(* CoDeSys 2.3.9.42 project: CR0451 AGV.pro *)
(* Libraries: ifm_PDMsmart_util_V010007.lib 26.10.09 12:29:10, ifm_RAWCan\ifm_RAWCan_NT_V020004.lib 3.11.15 19:07:52, ifm_J1939_NT\ifm_J1939_NT_V020004.lib 18.9.14 16:13:02, Util.lib 6.11.07 16:39:24, SysLibPlcCtrl.lib 13.6.03 15:49:00, SysLibFile.lib 23.9.04 10:11:36, SysLibTime.lib 27.4.05 10:36:52, LinuxSystemLib.Lib 18.3.03 13:26:50, ifm_pdm_file_V010006.lib 14.1.08 14:21:32, standard.lib 4.10.05 11:14:46, SysLibVisuBasicDisplay.lib 22.3.17 09:59:30, SysLibTargetVisu.lib 5.4.04 13:31:00, SysLibCallback.lib 26.9.08 17:43:52, ifm_CR0451_callback_visu.lib 22.3.17 09:59:30, SysLibStr.lib 13.6.03 15:49:00, ifm_CR0451\ifm_CR0451_Init_V030000.lib 22.3.17 09:59:30 *)

(* PLC configuration (modules and I/O channels)
Device Configuration [LocalConfiguration] node 0, in %IB0 out %QB0 {IFM_PARAM_WORD_TIME = 10}
KEY_F1 AT %IB0 [ChInputBool] F1 Key
KEY_F2 AT %IB1 [ChInputBool] F2 Key
KEY_F3 AT %IB2 [ChInputBool] F3 Key
KEY_F4 AT %IB3 [ChInputBool] F4 Key
KEY_UP AT %IB4 [ChInputBool] Up Key
KEY_DOWN AT %IB5 [ChInputBool] Down Key
KEY_LEFT AT %IB6 [ChInputBool] Left Key
KEY_RIGHT AT %IB7 [ChInputBool] Right Key
KEY_OK AT %IB8 [ChInputBool] Ok Key
RT_F1 AT %IB9 [ChInputBool] Rising Edge F1 Key
RT_F2 AT %IB10 [ChInputBool] Rising Edge F2 Key
RT_F3 AT %IB11 [ChInputBool] Rising Edge F3 Key
RT_F4 AT %IB12 [ChInputBool] Rising Edge F4 Key
RT_UP AT %IB13 [ChInputBool] Rising Edge Up Key
RT_DOWN AT %IB14 [ChInputBool] Rising Edge Down Key
RT_LEFT AT %IB15 [ChInputBool] Rising Edge Left Key
RT_RIGHT AT %IB16 [ChInputBool] Rising Edge Right Key
RT_OK AT %IB17 [ChInputBool] Rising Edge Ok Key
FT_F1 AT %IB18 [ChInputBool] Falling Edge F1 Key
FT_F2 AT %IB19 [ChInputBool] Falling Edge F2 Key
FT_F3 AT %IB20 [ChInputBool] Falling Edge F3 Key
FT_F4 AT %IB21 [ChInputBool] Falling Edge F4 Key
FT_UP AT %IB22 [ChInputBool] Falling Edge Up Key
FT_DOWN AT %IB23 [ChInputBool] Falling Edge Down Key
FT_LEFT AT %IB24 [ChInputBool] Falling Edge Left Key
FT_RIGHT AT %IB25 [ChInputBool] Falling Edge Right Key
FT_OK AT %IB26 [ChInputBool] Falling Edge Ok Key
Key Events [KeyEvents] node 3, in %IB27 out %QB0
  KEY_CHANGED AT %IB27 [ChInputBool] Event: Key Changed
  KEY_PRESSED AT %IB28 [ChInputBool] Event: Key is pressed
SUPPLY_VOLTAGE_VBBS AT %IW15 [ChInputWord] Supply voltage VBBS
SUPPLY_VOLTAGE_VU AT %IW16 [ChInputWord] Supply voltage VU
TEMPERATURE AT %IW17 [ChInputInt] Temperature
SCREEN_BACKLIGHT_CTRL AT %QB0 [ChOutputByte] Screen Backlight (0 - 100%)
KEY_BACKLIGHT_CTRL AT %QB1 [ChOutputByte] Key Backlight (0 - 100%)
CANopen Interface [CAN_OPEN] node 0, in %IB36 out %QB2
J1939 Interface [CAN_J1939] node 1, in %IB36 out %QB2
*)

(* Global variable list: Variables_Globales *)
VAR_GLOBAL

(* var for page and item menu selection *)
	menu_glob: INT:=1;
	PageIntern: WORD;
	Actual_Page: WORD;
  menu_item: ARRAY [0..20] OF BOOL;



END_VAR

VAR_GLOBAL RETAIN

END_VAR

(* POU PLC_PRG, ST *)
PROGRAM PLC_PRG
VAR
      xInitPageControl: BOOL;
	Shift_on_page_P00100: Shift_on_page_P00xxx;
	Shift_on_page_P00101: Shift_on_page_P00xxx;
	Shift_on_page_P00102: Shift_on_page_P00xxx;
	Shift_on_page_P00103: Shift_on_page_P00xxx;
	CAN_ENABLE_CAN1: CAN_ENABLE;
END_VAR
(* -++++++++++++++++-hieronder kun je het CAN channel activeren met   CAN_ENABLE  en/of  J1939_ENABLE-++++++++*)
CAN_ENABLE_CAN1(ENABLE:=TRUE, CHANNEL:= 1, BAUDRATE:=500 , RESULT=> );


(*++++++++++++++++++++++++++++++++++++++++++++++++++++++++++++++++++++++++++++++++++++++++++*)
(* -------------------------------------------initialiseren van het display CR0451---------------------------------------------------------------- *)
BasicDisplay_Init();
PDM_PAGECONTROL(
	INIT:= xInitPageControl,
	INIT_PAGE:=00001 ,
	PAGE_UP:= ,
	PAGE_DOWN:= ,
	PAGE_EXTERN:=PageIntern ,
	PAGE_MAX:=00108 ,                       (* de "hoogste pagina nummer opgeven*)
	BASENAME:='P',
	ACT_PAGE=>Actual_Page );

xInitPageControl:=FALSE;  (* pdm_pagecontrol moet slechts 1 keer worden uitgevoerd bij opstart, daarom init onmiddellijk op False gezet *)

(* startpagina en achterliggende pagina's beheren *)
(* zie eigen aangemaakte functieblok  Shift_on_pageP00XX,  de actuele pagina en het aantal menu items opgeven *)
Select_pages_on_mainpage();
Shift_on_page_P00100(Act_Page:= 00100, max_menu_items:=4);
Shift_on_page_P00101(Act_Page:= 00101, max_menu_items:= 4);
Shift_on_page_P00102(Act_Page:= 00102, max_menu_items:= 4);
Shift_on_page_P00103(Act_Page:= 00103, max_menu_items:= 3);

Return_main_next_page();    (* op iedere pagina, behalve de startpagina kan men naar volgende en vorige pagina gaan met de  F1 en F4  *)

(*-----------------------------------------------------------------------------------------------------------------------------------------------------*)

CAN_versturen_keys();

(*Programma verantwoordelijk voor het sturen van de modus van de AGV*)
ModusAGV();

ARDUINO_REC_POZXY();
ARDUINO_REC_US();
ARDUINO_REC_GYRO_BNO055();
END_PROGRAM

(* POU Shift_on_page_P00xxx, ST *)
FUNCTION_BLOCK Shift_on_page_P00xxx
VAR_INPUT
	Act_Page: INT;
	max_menu_items: INT;
END_VAR
VAR_OUTPUT
END_VAR
VAR
	menu_counter: INT;
	loop_counter: INT;
END_VAR
(*--------------------------------- WIJZIG NIETS AAN DEZE PROGRAMMA CODE--------------------------------------- *)
(*------  onderstaande code is toepasbaar op alle pagina's en laat toe met de UP en DOWN toetsen
te navigeren tussen de menu items --------------------------------------------------------------------------------------------*)
(* dit is functieblok met 2 inputs:  de pagina en het aantal MAXIMUM menu items moet opgegeven worden om de functieblok toe te passen *)

IF Actual_Page = Act_Page  THEN

IF RT_UP THEN
	 menu_counter:=menu_counter-1;
    	IF menu_counter<1 THEN
    	menu_counter:=1;
    	END_IF;
END_IF;
IF RT_DOWN  THEN
    menu_counter:=menu_counter+1;
    	IF menu_counter>max_menu_items THEN
    	menu_counter:=max_menu_items;
    	END_IF;
END_IF;

FOR loop_counter := 1 TO max_menu_items DO
IF loop_counter= menu_counter THEN
menu_item[menu_counter]:= TRUE;
ELSE
menu_item[loop_counter]:= FALSE;
END_IF
END_FOR
loop_counter:=1;

END_IF
END_FUNCTION_BLOCK

(* POU Select_pages_on_mainpage, ST *)
PROGRAM Select_pages_on_mainpage
VAR
END_VAR
(*--------------------------------- WIJZIG NIETS AAN DEZE PROGRAMMA CODE--------------------------------------------------- *)
(* dit programma zorgt ervoor dat je vanauit de startpagina P00100 kunt navigeren naar achterliggende pagina's*)

IF Actual_page=00100 THEN

IF menu_item[1]=TRUE AND RT_OK=TRUE THEN
	  menu_glob:=2;
      PageIntern:=00101;
END_IF;
(**********************************************************************************************)
IF menu_item[2]=TRUE  AND RT_OK=TRUE THEN
     menu_glob:=3;
      PageIntern:=00102;
END_IF;
(**********************************************************************************************)

IF menu_item[3]=TRUE AND RT_OK=TRUE THEN
	  menu_glob:=4;
      PageIntern:=00103;
END_IF;
(**********************************************************************************************)
(*
IF menu_item[4]=TRUE AND RT_OK=TRUE THEN 
	  menu_glob:=5;
      PageIntern:=00104;
END_IF;

enzovoort
*)



END_IF;
END_PROGRAM

(* POU Return_main_next_page, ST *)
PROGRAM Return_main_next_page
VAR

END_VAR
(*--------------------------------- WIJZIG NIETS AAN DEZE PROGRAMMA CODE--------------------------------------- *)
(* met onderstaand programma kun je vanaf elke pagina, behalve de startpagina P00100
met de toetsen F1 en F4 naar voorgaande of volgende pagina navigeren-----------------------------------------*)

IF RT_F1 = TRUE AND actual_page <> 00100 THEN (* if F1 is pressed return prev page *)
		menu_glob:=menu_glob-1;

  IF menu_glob<1 THEN
	  menu_glob:=1;
  END_IF;
END_IF;

IF RT_F4 = TRUE AND actual_page <> 00100 THEN  (* if F4 is pressed next page *)
 	menu_glob:=menu_glob+1;

  IF menu_glob >4 THEN  (* > 8 ingeval tot P00107 *)
   menu_glob:=1;
   END_IF;
END_IF


CASE menu_glob OF
1 : PageIntern:=00100;
2 : PageIntern:=00101;
3 : PageIntern:=00102;
4 : PageIntern:=00103;
(*
5 : PageIntern:=00104;
6 : PageIntern:=00105;
7 : PageIntern:=00106;
8 : PageIntern:=00107;
*)
END_CASE
END_PROGRAM

(* POU CAN_versturen_keys, ST *)
PROGRAM CAN_versturen_keys
VAR
	CAN_TX_ENH_CYCLIC_Keys: CAN_TX_ENH_CYCLIC;
END_VAR
CAN_TX_ENH_CYCLIC_Keys(
	ENABLE:=TRUE ,
	CHANNEL:=1 ,
	ID:=16#190 ,
	Extended:=FALSE ,
	DataLengthCode:=8 ,
	DATA:= , 
	PERIOD:= T#100ms,
	RESULT=> );

CAN_TX_ENH_CYCLIC_Keys.DATA[0]:=PACK(
	KEY_F1,
	KEY_F2,
	KEY_F3,
	KEY_F4,
	0,
	0,
	0,
	0);
END_PROGRAM

(* POU ModusAGV, ST *)
PROGRAM ModusAGV
VAR
	Manueel: BOOL := FALSE;
	Leren: BOOL;
	Automatisch: BOOL;
	CAN_TX_ENH_CYCLIC_ModusAGV: CAN_TX_ENH_CYCLIC;
END_VAR
(*We zitten op de pagina voor het kiezen van de modus van de AGV.
We hebben de keuze tussen manueel, leren en automatisch*)
(*OPM: Indien je een andere modus selecteert moet je op F3 drukken zodat de vorige op FALSE komt te staan
Het is ook niet mogelijk meerdere modussen tegelijk aan te zetten *)
IF Actual_page = 00101 THEN
	IF menu_item[1]= TRUE AND KEY_OK = TRUE  AND KEY_PRESSED = TRUE AND Leren = FALSE AND Automatisch = FALSE
	THEN
	Manueel := TRUE;
	ELSIF menu_item[2]= TRUE AND KEY_OK = TRUE AND KEY_PRESSED = TRUE AND Manueel = FALSE AND Automatisch = FALSE
	THEN
	Leren := TRUE;
	ELSIF menu_item[3]= TRUE AND KEY_OK = TRUE  AND KEY_PRESSED = TRUE AND Leren = FALSE AND Manueel = FALSE
	THEN
	Automatisch := TRUE;
	ELSIF KEY_F3 = TRUE
	THEN
	Manueel := FALSE;
	Leren := FALSE;
	Automatisch := FALSE;
	END_IF

END_IF

CAN_TX_ENH_CYCLIC_ModusAGV(
	ENABLE					:= TRUE,
	CHANNEL					:= 1 ,
	ID							:= 16#191 ,
	Extended					:= FALSE,
	DataLengthCode			:=1 ,
	DATA						:= ,
	PERIOD					:= t#100ms ,
	RESULT					=> );

CAN_TX_ENH_CYCLIC_ModusAGV.DATA[0]:= PACK(
	Manueel,
	Leren,
	Automatisch,
	0,
	0,
	0,
	0,
	0);
END_PROGRAM

(* POU ARDUINO_REC_POZXY, ST *)
PROGRAM ARDUINO_REC_POZXY
VAR
	CAN_RX_POZXY_COORD: CAN_RX;
	ARRAY_TO_DWORD_Xcoor: ARRAY_TO_DWORD;
	ARRAY_TO_DWORD_Ycoor: ARRAY_TO_DWORD;
END_VAR
CAN_RX_POZXY_COORD(
	ENABLE:= TRUE,
	CHANNEL:=1 ,
	ID:=16#A1 ,
	DATA=> , 
	RESULT=> );

IF  CAN_RX_POZXY_COORD.RESULT=1 THEN


ARRAY_TO_DWORD_Xcoor(
	Byte_0:=CAN_RX_POZXY_COORD.DATA[0] ,
	Byte_1:=CAN_RX_POZXY_COORD.DATA[1] ,
	Byte_2:=CAN_RX_POZXY_COORD.DATA[2] ,
	Byte_3:=CAN_RX_POZXY_COORD.DATA[3] ,
	DWORD_OUT=> );

ARRAY_TO_DWORD_Ycoor(
	Byte_0:=CAN_RX_POZXY_COORD.DATA[4] ,
	Byte_1:=CAN_RX_POZXY_COORD.DATA[5] ,
	Byte_2:=CAN_RX_POZXY_COORD.DATA[6] ,
	Byte_3:=CAN_RX_POZXY_COORD.DATA[7] ,
	DWORD_OUT=> );

END_IF
END_PROGRAM

(* POU ARDUINO_REC_US, ST *)
PROGRAM ARDUINO_REC_US
VAR
	CAN_RX_USranger: CAN_RX;
	wAfstand_US_ranger: WORD;
	ARRAY_TO_WORD_US: ARRAY_TO_WORD;
END_VAR
CAN_RX_USranger(
	ENABLE:=TRUE ,
	CHANNEL:=1 ,
	ID:=16#C1 ,
	DATA=> ,
	RESULT=> );

IF  CAN_RX_USranger.RESULT = 1 THEN

ARRAY_TO_WORD_US(Byte_0:=CAN_RX_USranger.DATA[0] , Byte_1:=CAN_RX_USranger.DATA[1] , WORD_OUT=>wAfstand_US_ranger );



END_IF
END_PROGRAM

(* POU ARDUINO_REC_GYRO_BNO055, ST *)
PROGRAM ARDUINO_REC_GYRO_BNO055
VAR
	CAN_RX_BNO055: CAN_RX;
	ARRAY_TO_DWORD_X_DIR: ARRAY_TO_DWORD;
END_VAR
CAN_RX_BNO055(
	ENABLE:=TRUE ,
	CHANNEL:=1 ,
	ID:=16#B1 ,
	DATA=> , 
	RESULT=> );

IF CAN_RX_BNO055.RESULT=1 THEN

ARRAY_TO_DWORD_X_DIR(
	Byte_0:=CAN_RX_BNO055.DATA[0] ,
	Byte_1:=CAN_RX_BNO055.DATA[1] ,
	Byte_2:=CAN_RX_BNO055.DATA[2] ,
	Byte_3:=CAN_RX_BNO055.DATA[3] ,
	DWORD_OUT=> );



END_IF
END_PROGRAM

(* Visualisation PAGE_SELECT/P00100
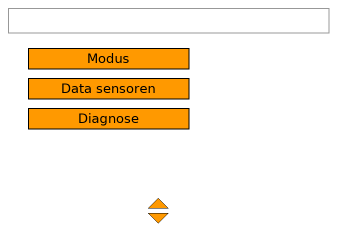
rectangle at (0,0)-(321,25): text "MENU"
rectangle at (20,70)-(181,91): text "Data sensoren"; alarm colour if .menu_item[2]
rectangle at (20,40)-(181,61): text "Modus"; alarm colour if .menu_item[1]
rectangle at (20,100)-(181,121): text "Diagnose"; alarm colour if .menu_item[3]
rectangle at (30,190)-(136,211): text "navigeer met"
rectangle at (160,190)-(306,211): text "en bevestig met OK"
2 more shapes without text or variables
*)

(* Visualisation PAGE_SELECT/P00101
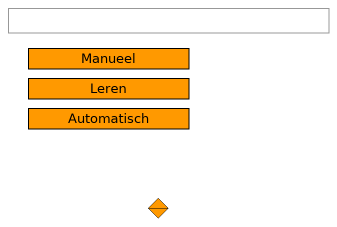
rectangle at (0,0)-(321,25): text "MODUS"
rectangle at (20,40)-(181,61): text "Manueel"; alarm colour if .menu_item[1]
rectangle at (20,70)-(181,91): text "Leren"; alarm colour if .menu_item[2]
rectangle at (20,100)-(181,121): text "Automatisch"; alarm colour if .menu_item[3]
rectangle at (30,190)-(136,211): text "navigeer met"
rectangle at (160,190)-(306,211): text "en bevestig met OK"
2 more shapes without text or variables
*)

(* Visualisation PAGE_SELECT/P00102
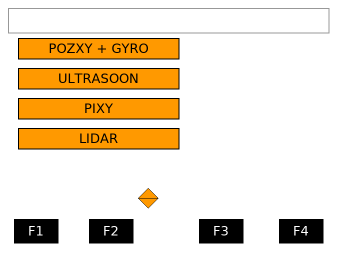
rectangle at (10,30)-(171,51): text "POZXY + GYRO"; alarm colour if .menu_item[1]
rectangle at (10,60)-(171,81): text "ULTRASOON"; alarm colour if .menu_item[2]
rectangle at (0,0)-(321,25): text "ARDUINO SENSOREN"
rectangle at (20,180)-(126,201): text "navigeer met"
rectangle at (150,180)-(296,201): text "en bevestig met OK"
rectangle at (10,90)-(171,111): text "PIXY"; alarm colour if .menu_item[3]
rectangle at (5,210)-(51,236): text "F1"
rectangle at (80,210)-(126,236): text "F2"
rectangle at (270,210)-(316,236): text "F4"
rectangle at (190,210)-(236,236): text "F3"
rectangle at (10,120)-(171,141): text "LIDAR"; alarm colour if .menu_item[4]
2 more shapes without text or variables
*)

(* Visualisation PAGE_SELECT/P00103
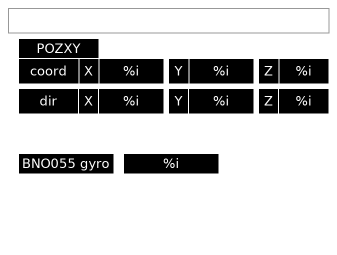
rectangle at (10,30)-(91,51): text "POZXY"
rectangle at (-1,219)-(40,240): text "<<<"
rectangle at (274,219)-(320,240): text ">>>"
rectangle at (0,0)-(321,25): text "ARDUINO SENSOREN"
rectangle at (90,50)-(156,76): text "%i"; shows ARDUINO_REC_POZXY.ARRAY_TO_DWORD_Xcoor.DWORD_OUT
rectangle at (180,50)-(246,76): text "%i"; shows ARDUINO_REC_POZXY.ARRAY_TO_DWORD_Ycoor.DWORD_OUT
rectangle at (270,50)-(321,76): text "%i"
rectangle at (70,50)-(91,76): text "X"
rectangle at (160,50)-(181,76): text "Y"
rectangle at (250,50)-(271,76): text "Z"
rectangle at (10,145)-(106,166): text "BNO055 gyro"
rectangle at (10,50)-(71,76): text "coord"
rectangle at (10,80)-(71,106): text "dir"
rectangle at (250,80)-(271,106): text "Z"
rectangle at (160,80)-(181,106): text "Y"
rectangle at (70,80)-(91,106): text "X"
rectangle at (270,80)-(321,106): text "%i"
rectangle at (180,80)-(246,106): text "%i"
rectangle at (90,80)-(156,106): text "%i"
rectangle at (115,145)-(211,166): text "%i"; shows ARDUINO_REC_GYRO_BNO055.ARRAY_TO_DWORD_X_DIR.DWORD_OUT
*)
